(* IEC 61131-3 sources: Industry-PLC-LLM/data/PLCBEAD_repo/PLCBEAD_PLCEmbed-main/PLC-BEAD/Source/GEB/SETUP_HOLIDAY_FR, 1 file *)

(* ---- SETUP_HOLIDAY_FR.ST ---- *)
TYPE oscat_HOLIDAY_DATA :
	STRUCT
		NAME : STRING;
		DAY  : SINT;
		MONTH : SINT;
		USE : SINT;
		PAD_BYTE : BYTE;
	END_STRUCT;
END_TYPE

TYPE
	oscat_HOLIDAY_DATA_0_29 	: ARRAY [0..29] OF oscat_HOLIDAY_DATA;
END_TYPE

FUNCTION_BLOCK SETUP_HOLIDAY_FR_Block

	VAR_IN_OUT
		HD :	oscat_HOLIDAY_DATA_0_29;
	END_VAR

	VAR
		init :	BOOL;
	END_VAR

	IF init THEN RETURN; END_IF;

	init := TRUE;

	HD[00].NAME := 'Nouve an';
	HD[00].DAY   := SINT#01;
	HD[00].MONTH := SINT#01;
	HD[00].USE := SINT#01;

	HD[01].NAME := 'St Valentin';
	HD[01].DAY   := SINT#14;
	HD[01].MONTH := SINT#02;
	HD[01].USE := SINT#00;

	HD[02].NAME := 'Vendredi Saint (alsace)';
	HD[02].DAY   := SINT#-2;
	HD[02].MONTH := SINT#00;
	HD[02].USE := SINT#00;

	HD[03].NAME := 'Dimanche de pques';
	HD[03].DAY   := SINT#00;
	HD[03].MONTH := SINT#00;
	HD[03].USE := SINT#01;

	HD[04].NAME := 'Lundi de pques';
	HD[04].DAY   := SINT#01;
	HD[04].MONTH := SINT#00;
	HD[04].USE := SINT#01;

	HD[05].NAME := 'Jeudi de Ascension';
	HD[05].DAY   := SINT#39;
	HD[05].MONTH := SINT#00;
	HD[05].USE := SINT#01;

	HD[06].NAME := 'dimanche de Pentecte';
	HD[06].DAY   := SINT#49;
	HD[06].MONTH := SINT#00;
	HD[06].USE := SINT#01;

	HD[07].NAME := 'jeudi de la Trinit';
	HD[07].DAY   := SINT#60;
	HD[07].MONTH := SINT#00;
	HD[07].USE := SINT#00;

	HD[08].NAME := 'Fte du travail';
	HD[08].DAY   := SINT#01;
	HD[08].MONTH := SINT#05;
	HD[08].USE := SINT#01;

	HD[09].NAME := 'Victoire 1945 ';
	HD[09].DAY   := SINT#08;
	HD[09].MONTH := SINT#05;
	HD[09].USE := SINT#01;

	HD[10].NAME := 'Prise de La bastille';
	HD[10].DAY   := SINT#14;
	HD[10].MONTH := SINT#07;
	HD[10].USE := SINT#01;

	HD[11].NAME := '15 Aot 1944';
	HD[11].DAY   := SINT#15;
	HD[11].MONTH := SINT#08;
	HD[11].USE := SINT#01;

	HD[12].NAME := 'Halloween';
	HD[12].DAY   := SINT#31;
	HD[12].MONTH := SINT#10;
	HD[12].USE := SINT#00;

	HD[13].NAME := 'Armistice 1918';
	HD[13].DAY   := SINT#11;
	HD[13].MONTH := SINT#11;
	HD[13].USE := SINT#01;

	HD[14].NAME := 'Nol';
	HD[14].DAY   := SINT#25;
	HD[14].MONTH := SINT#12;
	HD[14].USE := SINT#01;

	HD[15].NAME := 'Saint tienne (alsace)';
	HD[15].DAY   := SINT#26;
	HD[15].MONTH := SINT#12;
	HD[15].USE := SINT#00;

	HD[16].NAME := 'Fte de la musique';
	HD[16].DAY   := SINT#21;
	HD[16].MONTH := SINT#06;
	HD[16].USE := SINT#00;
END_FUNCTION_BLOCK

PROGRAM program0
  VAR
    LocalVar0 : oscat_HOLIDAY_DATA_0_29;
	func_block : SETUP_HOLIDAY_FR_Block;
  END_VAR
	func_block.HD  := LocalVar0;
	func_block();
	LocalVar0 := func_block.HD;
END_PROGRAM
